(* IEC 61131-3 sources: st2cpp/examples/processImage, 1 file *)

(* ---- test_process_image.st ---- *)
(*
* test_process_image.st
* Test file for Process Image functionality
* Tests: %I, %Q, %M addresses with different qualifiers and placeholders "*"
*)

TYPE TestEnum :
    (
    IDLE,
    RUNNING,
    STOPPED,
    ERROR
    );
END_TYPE

TYPE MotorStatus :
    STRUCT
        Running : BOOL;
        Speed : INT;
        Temp : REAL;
        Fault : BOOL;
    END_STRUCT;
END_TYPE

(* Global variables with AT addresses - fixed and placeholder *)
VAR_GLOBAL
    (* Fixed addresses - will be marked as occupied *)
    StartButton AT %IX0.0 : BOOL := FALSE;
    StopButton AT %IX0.1 : BOOL := FALSE;
    Emergency AT %IX0.2 : BOOL := FALSE;

    MotorOutput AT %QX0.0 : BOOL := FALSE;
    AlarmLight AT %QX0.1 : BOOL := FALSE;
    StatusWord AT %QW2 : WORD := 16#0000;

    Counter AT %MW10 : INT := 0;
    Temperature AT %MW12 : INT := 25;
    Flags AT %MB20 : BYTE := 0;
    Status AT %ML22 : DWORD := 0;

    (* ========== PLACEHOLDER ADDRESSES - auto-allocated ========== *)

    (* BIT placeholders - will be allocated after fixed bits *)
    SensorA AT %IX* : BOOL := FALSE;       (* Will be allocated automatically *)
    SensorB AT %IX* : BOOL := FALSE;       (* Will be allocated automatically *)
    ActuatorA AT %QX* : BOOL := FALSE;     (* Will be allocated automatically *)
    ActuatorB AT %QX* : BOOL := FALSE;     (* Will be allocated automatically *)
    FlagA AT %MX* : BOOL := FALSE;         (* Will be allocated automatically *)

    (* BYTE placeholders - aligned to byte boundaries *)
    AnalogInput AT %IB* : BYTE := 0;       (* Will be allocated to %IB1 (after fixed bits) *)
    AnalogOutput AT %QB* : BYTE := 0;      (* Will be allocated automatically *)
    StatusFlags AT %MB* : BYTE := 0;       (* Will be allocated automatically *)

    (* WORD placeholders - must be aligned to 2-byte boundary *)
    Setpoint AT %IW* : INT := 100;         (* Will be allocated automatically *)
    Feedback AT %IW* : INT := 0;           (* Will be allocated automatically *)
    Command AT %QW* : WORD := 16#0000;     (* Will be allocated automatically *)
    MarkerData AT %MW* : WORD := 0;        (* Will be allocated automatically *)

    (* DWORD placeholders - must be aligned to 4-byte boundary *)
    LargeCounter AT %MD* : DWORD := 0;     (* Will be allocated automatically *)
    Timestamp AT %MD* : DWORD := 0;        (* Will be allocated automatically *)

    (* Mixed placeholders in different areas *)
    DiagDWord AT %MD* : DWORD := 0;       (* Will be allocated automatically *)
    DebugFlag AT %MX* : BOOL := FALSE;     (* Will be allocated automatically *)
    DebugValue AT %MW* : INT := 0;         (* Will be allocated automatically *)
END_VAR

(* Function block with process image access and methods *)
FUNCTION_BLOCK MotorController
    VAR_INPUT
        Enable : BOOL;
        Speed : INT;
    END_VAR

    VAR_OUTPUT
        Running : BOOL;
        Fault : BOOL;
    END_VAR

    VAR
        Timer : INT := 0;
        (* Local AT placeholder inside FB *)
        InternalFlag AT %MX* : BOOL := FALSE;  (* Will be allocated automatically *)
        InternalData AT %MW* : INT := 0;       (* Will be allocated automatically *)
    END_VAR

    METHOD CheckOverheat : BOOL
        VAR_INPUT
            Temp : INT;
        END_VAR
        VAR_OUTPUT
            Overheat : BOOL;
        END_VAR
        Overheat := Temp > 80;
        CheckOverheat := Overheat;
    END_METHOD

    METHOD ReadInternalData : INT
        VAR_OUTPUT
            Value : INT;
        END_VAR
        Value := InternalData;
    END_METHOD
END_FUNCTION_BLOCK

(* Main program - NO methods allowed! *)
PROGRAM Main
    VAR
        Motor : MotorController;
        TempRead : INT;
        State : TestEnum := TestEnum.IDLE;
        Status : MotorStatus;
        CycleCounter : INT := 0;
        NewState : TestEnum := IDLE;
        Updated : BOOL := FALSE;
        Start : BOOL := FALSE;
        Stop : BOOL := FALSE;
        EStop : BOOL := FALSE;
        Increment : BOOL := FALSE;
        NewTemp : INT := 0;
        (* Local AT placeholders inside program *)
        LocalSensor AT %IX* : BOOL := FALSE;   (* Will be allocated automatically *)
        LocalOutput AT %QX* : BOOL := FALSE;   (* Will be allocated automatically *)
        LocalData AT %MW* : INT := 0;          (* Will be allocated automatically *)
    END_VAR

    (* Main program body *)
    (* Read inputs *)
    Start := StartButton;
    Stop := StopButton;
    EStop := Emergency;

    (* Check emergency *)
    IF Emergency THEN
        MotorOutput := FALSE;
        AlarmLight := TRUE;
        Flags := Flags OR INT_TO_BYTE(16#80);
    END_IF;

    (* Update outputs based on state *)
    IF NOT Emergency THEN
        IF State = TestEnum.RUNNING THEN
            MotorOutput := TRUE;
            AlarmLight := FALSE;
            StatusWord := INT_TO_WORD(16#0001);
        ELSIF State = TestEnum.STOPPED THEN
            MotorOutput := FALSE;
            AlarmLight := TRUE;
            StatusWord := INT_TO_WORD(16#0002);
        ELSE
            MotorOutput := FALSE;
            AlarmLight := FALSE;
            StatusWord := INT_TO_WORD(16#0000);
        END_IF;
    END_IF;

    (* Process counter *)
    IF Increment THEN
        Counter := Counter + 1;
    END_IF;

    (* Update temperature *)
    Temperature := NewTemp;
    Status.Temp := INT_TO_REAL(NewTemp) / 10.0;

    (* Use the function block *)
    Motor(Enable := Start, Speed := 100);

    (* Update status *)
    Updated := TRUE;

    (* Use local AT variables *)
    LocalSensor := SensorA;
    LocalOutput := ActuatorA;
    LocalData := Setpoint;
END_PROGRAM

(* Another program with different AT address patterns - NO methods! *)
PROGRAM Diagnostic
    VAR
        ErrorCode AT %MW50 : INT := 0;
        ErrorTime AT %MD52 : DWORD := 0;
        ErrorFlag AT %MX54.0 : BOOL := FALSE;
        Status AT %MW60 : INT := 0;
        Code : INT := 0;
        (* Local AT placeholders inside Diagnostic program *)
        DiagData AT %MD* : DWORD := 0;         (* Will be allocated automatically *)
        DiagFlag AT %MX* : BOOL := FALSE;      (* Will be allocated automatically *)
        DiagWord AT %MW* : WORD := 0;          (* Will be allocated automatically *)
    END_VAR

    (* Set error *)
    ErrorCode := Code;
    ErrorTime := INT_TO_DWORD(0);
    ErrorFlag := TRUE;
    Status := 1;

    (* Clear error *)
    ErrorCode := 0;
    ErrorTime := INT_TO_DWORD(0);
    ErrorFlag := FALSE;
    Status := 0;

    (* Use placeholders *)
    DiagData := ErrorTime;
    DiagFlag := ErrorFlag;
    DiagWord := INT_TO_WORD(16#FFFF);
END_PROGRAM

(* Function that uses process image addresses - fixed and placeholder *)
FUNCTION GetMotorSpeed : INT
    VAR_INPUT
        MotorID : INT;
    END_VAR
    VAR
        Speed AT %IW100 : INT := 0;
        Speed2 AT %IW102 : INT := 0;
        (* Local AT placeholders inside function *)
        TempSpeed AT %IW* : INT := 0;          (* Will be allocated automatically *)
        SensorValue AT %IW* : INT := 0;        (* Will be allocated automatically *)
    END_VAR
    (* Read speed from input addresses *)
    IF MotorID = 1 THEN
        GetMotorSpeed := Speed;
    ELSE
        GetMotorSpeed := Speed2;
    END_IF;
END_FUNCTION
